FUNCTION_BLOCK FB_ExtractString
VAR_INPUT
END_VAR
VAR_OUTPUT
END_VAR
VAR
END_VAR

END_FUNCTION_BLOCK

(* stored: Version 1.1.0.1
   POU FB_ExtractString: Id {85391f85-6b56-41db-91af-59cb7cf4ebc2}, SpecialFunc None *)
